                               // Determine distance for positioning command (relative)
                               IF (#configuration.jog.mode = #JOG_MODE_NEW_INCREMENT) // In this mode a new increment is always set
                                 OR ((#configuration.jog.mode = #JOG_MODE_CONTINUE_INCREMENT) AND (#statResetIncJog = TRUE))
                               THEN
                                 #statResetIncJog := FALSE;
                                 // New increment
                                 #statIncJogStartPosition := "LAxisCtrl_UnpubAxisPosition"(#statAxis); // Targetposition for increment
                                 #statIncrement := ABS(#configuration.jog.increment); // absolute Distance for increment
                                 IF (#statBasicCommand.%X2 = TRUE) THEN
                                   // JogForward selected
                                   #statPosition := ABS(#configuration.jog.increment);
                                   #statIncrement := #statPosition;
                                   #statIncJogDirectionOld := #FORWARD_DIR;
                                 ELSIF (#statBasicCommand.%X3 = TRUE) THEN
                                   // JogBackward selected
                                   #statPosition := - ABS(#configuration.jog.increment);
                                   #statIncrement := #statPosition;
                                   #statIncJogDirectionOld := #BACKWARD_DIR;
                                 ELSE
                                   // Normal not possible to reach ELSE-branch
                                   #statIncJogDirectionOld := 0;
                                 END_IF;
                               ELSE
                                 // Check for modulo axis
                                 IF ("LAxisCtrl_UnpubAxisModuloEnabled"(#statAxis) = FALSE) THEN
                                   // No Modulo enabled
                                   // Continue increment
                                   #statPosition := (#statIncJogStartPosition + #statIncrement) - "LAxisCtrl_UnpubAxisPosition"(#statAxis);
                                   // Distance   :=            setpoint                         - actualvalue
                                 ELSE
                                   // Modulo enabled
                                   #statPosition := #statIncJogDistance;
                                 END_IF;
                               END_IF;
                               #statIncJogSubState := #INC_JOG_START;

                               // Store Dynamics
                               #statBasicVelocity := ABS(#configuration.jog.velocity);
                               #statBasicAcceleration := #configuration.jog.acceleration;
                               #statBasicDeceleration := #configuration.jog.deceleration;
                               #statBasicJerk := #configuration.jog.jerk;
                             ELSE
                               // Errorhandling - Invalid direction (forward and backward selected)
                               #statStatus := #ERR_INVALID_JOG_DIR;
                               #statStatusText := STRING#'ERR_INVALID_JOG_DIR';
                               #statErrorAutoCleared := TRUE;
                               #statDiagnostics.subfunctionStatus := #statSubfunctionStatus := 0;
                               #statDiagnostics.basicMotionState := #statBasicMotionState;
                               // Set next state
                               #statFBState := #AXIS_STOP_ON_ERROR_SELECTION;
                               #statBasicMotionState := #NO_SELECTION;
                               #statExeOfBasicMotion := #CMD_ERROR;
                               #statIncJogSubState := #INC_JOG_IDLE;
                             END_IF;

                           ELSIF ((#statBasicCommand.%X2 = FALSE) AND (#statBasicCommand.%X3 = FALSE)) // No jog input selected --> Stop moving
                             AND (#statIncJogSubState <> #INC_JOG_STOP)
                           THEN
                             // Reset HALT command
                             #instHalt(Axis := #statAxis,
                                       Execute := FALSE);
                             #statIncJogSubState := #INC_JOG_STOP;
                             #statIncJogDistance := "LAxisCtrl_UnpubAxisPositioningDistance"(#statAxis);

                           ELSIF (#statBasicCommand.%X2 = TRUE) AND (#statBasicCommand.%X3 = TRUE) // jogForward and jogBackward selected - Error
                           THEN
                             // Reset HALT command
                             #instHalt(Axis := #statAxis,
                                       Execute := FALSE);
                             #statIncJogSubState := #INC_JOG_STOP;
                             // Errorhandling
                             #statStatus := #ERR_INVALID_JOG_DIR;
                             #statStatusText := STRING#'ERR_INVALID_JOG_DIR';
                             #statErrorAutoCleared := TRUE;
                             #statDiagnostics.subfunctionStatus := #statSubfunctionStatus := 0;
                             // Set next state
                             #statExeOfBasicMotion := #CMD_ERROR;
                             #statBasicMotionState := #NO_SELECTION;
                             #statFBState := #AXIS_STOP_ON_ERROR_SELECTION;
                           ELSE
                             ; // Command running
                           END_IF;

                           // Select motion
                           CASE #statIncJogSubState OF
                             #INC_JOG_IDLE:
                               ; // Do nothing - Error occurred (jogforward and jogbackward are set in firstCycle of operation)

                             #INC_JOG_START: // Run jog operation --> Motion stops automatically if increment complete
                               #instMoveRelative(Axis := #statAxis,
                                                 Execute := TRUE,
                                                 Distance := #statPosition,
                                                 Velocity := #statBasicVelocity,
                                                 Acceleration := #statBasicAcceleration,
                                                 Deceleration := #statBasicDeceleration,
                                                 Jerk := #statBasicJerk);

                               // Evaluate MC_Command
                               IF (#instMoveRelative.Done = TRUE) THEN
                                 // Increment completed
                                 #statResetIncJog := TRUE;
                                 // Set next state
                                 #statExeOfBasicMotion := #CMD_DONE;
                                 #statIncJogSubState := #INC_JOG_IDLE;

                               ELSIF (#instMoveRelative.Error = TRUE) THEN
                                 #statResetIncJog := TRUE;
                                 // Errorhandling
                                 #statStatus := #ERR_MC_MOVERELATIVE;
                                 #statStatusText := STRING#'ERR_MC_MOVERELATIVE';
                                 #statErrorAutoCleared := TRUE;
                                 #statDiagnostics.subfunctionStatus := #statSubfunctionStatus := #instMoveRelative.ErrorID;
                                 // Set next state
                                 #statFBState := #AXIS_STOP_ON_ERROR_SELECTION;
                                 #statBasicMotionState := #NO_SELECTION;
                                 #statExeOfBasicMotion := #CMD_ERROR;
                                 #statIncJogSubState := #INC_JOG_IDLE;

                               ELSIF (#instMoveRelative.CommandAborted = TRUE) THEN
                                 #statResetIncJog := TRUE;
                                 #statExeOfBasicMotion := #CMD_ABORTED;
                                 #statIncJogSubState := #INC_JOG_IDLE;
                               ELSE
                                 ; // Wait for next state
                               END_IF;

                             #INC_JOG_STOP: // Executed if inputs are reset --> Stop jog operation OR if jogForward and jogBackward are set --> Error and stop axis
                               #instHalt(Axis := #statAxis,
                                         Execute := TRUE,
                                         Deceleration := #statBasicDeceleration,
                                         AbortAcceleration := FALSE,
                                         Jerk := #statBasicJerk);

                               // Evaluate MC_Command
                               IF (#instHalt.Done = TRUE) THEN
                                 // Set next state
                                 #statExeOfBasicMotion := #CMD_END_PROCESS;
                                 #statIncJogSubState := #INC_JOG_IDLE;

                               ELSIF (#instHalt.Error = TRUE) THEN
                                 #statResetIncJog := TRUE;
                                 // Errorhandling
                                 #statStatus := #ERR_MC_HALT;
                                 #statStatusText := STRING#'ERR_MC_HALT';
                                 #statErrorAutoCleared := TRUE;
                                 #statDiagnostics.subfunctionStatus := #statSubfunctionStatus := #instHalt.ErrorID;
                                 // Set next state
                                 #statFBState := #AXIS_STOP_ON_ERROR_SELECTION;
                                 #statBasicMotionState := #NO_SELECTION;
                                 #statExeOfBasicMotion := #CMD_ERROR;
                                 #statIncJogSubState := #INC_JOG_IDLE;

                               ELSIF (#instHalt.CommandAborted = TRUE) THEN
                                 #statResetIncJog := TRUE;
                                 // Set next state
                                 #statIncJogSubState := #INC_JOG_IDLE;
                                 #statExeOfBasicMotion := #CMD_ABORTED;
                               ELSE
                                 ; // Wait for stopping axis
                               END_IF;
                             ELSE
                               // Errorhandling
                               #statStatus := #ERR_UNDEFINED_INCREMENTAL_JOG_SUBSTATE;
                               #statStatusText := STRING#'ERR_UNDEFINED_INCREMENTAL_JOG_SUBSTATE';
                               #statErrorUserCleared := TRUE;
                               #statDiagnostics.subfunctionStatus := #statSubfunctionStatus := 0;
                               // Set errorstate
                               #statFBState := #FB_ERROR;
                           END_CASE;

                         #CMD_DONE,
                         #CMD_ABORTED,
                         #CMD_ERROR,
                         #CMD_END_PROCESS:
                           // Return to NO_SELECTION if command finished
                           IF (#statBasicCommand.%X2 = FALSE) AND (#statBasicCommand.%X3 = FALSE)
                           THEN
                             // jogForward and jogbackward inputs are reset
                             #statExeOfBasicMotion := #CMD_BUSY;
                             #statBasicMotionState := #NO_SELECTION;
                           ELSE
                             ; // Wait for falling edge at inputs for jog
                           END_IF;
                         ELSE
                           // Errorhandling
                           #statStatus := #ERR_UNDEFINED_INCREMENTAL_JOG_STATE;
                           #statStatusText := STRING#'ERR_UNDEFINED_INCREMENTAL_JOG_STATE';
                           #statErrorUserCleared := TRUE;
                           #statDiagnostics.subfunctionStatus := #statSubfunctionStatus := 0;
                           #statDiagnostics.basicMotionState := #statBasicMotionState;
                           // Set errorstate
                           #statFBState := #FB_ERROR;
                       END_CASE;
                     END_REGION
                   ELSE
                     // Errorhandling - Invalid jog state
                     #statStatus := #ERR_INVALID_JOG_MODE;
                     #statStatusText := STRING#'#ERR_INVALID_JOG_MODE';
                     #statErrorAutoCleared := TRUE;
                     #statDiagnostics.subfunctionStatus := #statSubfunctionStatus := 0;
                     // Set next state
                     #statFBState := #AXIS_STOP_ON_ERROR_SELECTION;
                     #statBasicMotionState := #NO_SELECTION;
                 END_CASE;
               END_REGION

             #MOVE_VELOCITY_SELECTED:
               // Additional features (applicative): Change setpoint on the fly (Velocity) 
               REGION MOVEVELOCITY_SELECTED
                 // Firstcycle of command
                 IF (#statFirstCycleBasicMotion = TRUE) THEN
                   // Reset MC_MOVEVELOCITY command
                   #instMoveVelocity(Axis := #statAxis,
                                     Execute := FALSE);

                   #statVelocityChangeOnTheFly := #configuration.moveVelocity.velocityChangeOnTheFly;
                   #statBasicVelocity := #configuration.moveVelocity.velocity;                     // Store the last adjusted velocity value
                   #statBasicAcceleration := #configuration.moveVelocity.acceleration;             // Store the last adjusted acceleration value
                   #statBasicDeceleration := #configuration.moveVelocity.deceleration;             // Store the last adjusted deceleration value
                   #statBasicJerk := #configuration.moveVelocity.jerk;                             // Store the last adjusted jerk value 
                   #statDirection := #configuration.moveVelocity.direction;                        // Store the last adjusted axis direction 
                   #statPositionControlled := #configuration.moveVelocity.positionControlled;      // Store the last adjusted motion mode

                 ELSIF (#statVelocityChangeOnTheFly = TRUE) AND (#configuration.moveVelocity.velocity <> #statBasicVelocity) // Velocity changed
                   AND (#instMoveVelocity.CommandAborted = FALSE)
                 THEN
                   // Reset MC_MOVEVELOCITY command
                   #instMoveVelocity(Axis := #statAxis,
                                     Execute := FALSE);
                   #statBasicVelocity := #configuration.moveVelocity.velocity;                     // Store the last adjusted velocity value

                   // V1.0.5 Copy also dynamics
                   #statBasicAcceleration := #configuration.moveVelocity.acceleration;             // Store the last adjusted acceleration value
                   #statBasicDeceleration := #configuration.moveVelocity.deceleration;             // Store the last adjusted deceleration value
                   #statBasicJerk := #configuration.moveVelocity.jerk;                             // Store the last adjusted jerk value 
                   #statDirection := #configuration.moveVelocity.direction;                        // Store the last adjusted axis direction 
                   #statPositionControlled := #configuration.moveVelocity.positionControlled;      // Store the last adjusted motion mode
                 END_IF;

                 // Call MC_Command
                 #instMoveVelocity(Axis := #statAxis,
                                   Execute := #statBasicCommand.%X4 OR #statFirstCycleBasicMotion, // Input: moveVelocity
                                   Velocity := #statBasicVelocity,
                                   Acceleration := #statBasicAcceleration,
                                   Deceleration := #statBasicDeceleration,
                                   Jerk := #statBasicJerk,
                                   Direction := #statDirection,
                                   PositionControlled := #statPositionControlled,
                                   Current := FALSE);

                 // Evaluate MC_Command
                 IF (#instMoveVelocity.Busy = FALSE) AND
                   (#instMoveVelocity.Error = FALSE) AND
                   (#instMoveVelocity.CommandAborted = FALSE) AND
                   (#instMoveVelocity.InVelocity = FALSE)
                 THEN
                   // Return to NO_SELECTION if command finished
                   #statBasicMotionState := #NO_SELECTION;

                 ELSIF (#instMoveVelocity.Error = TRUE)
                 THEN
                   // Errorhandling
                   #statStatus := #ERR_MC_MOVEVELOCITY;
                   #statStatusText := STRING#'ERR_MC_MOVEVELOCITY';
                   #statErrorAutoCleared := TRUE;
                   #statDiagnostics.subfunctionStatus := #statSubfunctionStatus := #instMoveVelocity.ErrorID;
                   #statVelocityChangeOnTheFly := FALSE;
                   // Set next state
                   #statFBState := #AXIS_STOP_ON_ERROR_SELECTION;
                   #statBasicMotionState := #NO_SELECTION;
                 ELSE
                   ; // Command selected
                 END_IF;

                 // Write MC_Command outputs to internal variable
                 #statExeOfBasicMotion := 16#0;
                 #statExeOfBasicMotion.%X0 := #instMoveVelocity.Busy;
                 #statExeOfBasicMotion.%X2 := #instMoveVelocity.CommandAborted;
                 #statExeOfBasicMotion.%X3 := #instMoveVelocity.Error;
                 #statExeOfBasicMotion.%X4 := #instMoveVelocity.InVelocity;
               END_REGION

             #POS_RELATIVE_SELECTED:
               // Additional features (applicative): Specified direction
               REGION POS_RELATIVE_SELECTED
                 // Firstcycle of command
                 IF (#statFirstCycleBasicMotion = TRUE) THEN
                   // Configurate the direction of rotation
                   IF ((#configuration.posRelative.direction = 0) AND (#configuration.posRelative.distance >= 0.0)) // Sign of distance is evaluated
                     OR (#configuration.posRelative.direction = #FORWARD_DIR) // Forward direction
                   THEN
                     #statPosition := ABS(#configuration.posRelative.distance);
                     // Reset MC_MOVERELATIVE command
                     #instMoveRelative(Axis := #statAxis,
                                       Execute := FALSE);
                     #statApplicativeBasicMotionError := FALSE;

                   ELSIF ((#configuration.posRelative.direction = 0) AND (#configuration.posRelative.distance < 0.0)) // Sign of distance is evaluated
                     OR (#configuration.posRelative.direction = #BACKWARD_DIR) // Backward direction
                   THEN
                     #statPosition := - ABS(IN := #configuration.posRelative.distance);
                     // Reset MC_MOVERELATIVE command
                     #instMoveRelative(Axis := #statAxis,
                                       Execute := FALSE);
                     #statApplicativeBasicMotionError := FALSE;
                   ELSE
                     // Errorhandling - Invalid direction
                     #statStatus := #ERR_INVALID_POS_RELATIVE_DIR;
                     #statStatusText := STRING#'ERR_INVALID_POS_RELATIVE_DIR';
                     #statErrorAutoCleared := TRUE;
                     #statDiagnostics.subfunctionStatus := #statSubfunctionStatus := 0;
                     #statApplicativeBasicMotionError := TRUE;
                     // Set next state
                     #statFBState := #AXIS_STOP_ON_ERROR_SELECTION;
                     #statBasicMotionState := #NO_SELECTION;
                   END_IF;
                 END_IF;

                 IF (#statApplicativeBasicMotionError = FALSE) THEN
                   // Call MC_Command
                   #instMoveRelative(Axis := #statAxis,
                                     Execute := #statBasicCommand.%X5 OR #statFirstCycleBasicMotion, // Input: posRelative
                                     Distance := #statPosition,
                                     Velocity := #configuration.posRelative.velocity,
                                     Acceleration := #configuration.posRelative.acceleration,
                                     Deceleration := #configuration.posRelative.deceleration,
                                     Jerk := #configuration.posRelative.jerk);

                   // Evaluate MC_Command
                   IF (#instMoveRelative.Busy = FALSE) AND
                     (#instMoveRelative.Error = FALSE) AND
                     (#instMoveRelative.Done = FALSE) AND
                     (#instMoveRelative.CommandAborted = FALSE)
                   THEN
                     // Return to NO_SELECTION if command finished
                     #statBasicMotionState := #NO_SELECTION;

                   ELSIF (#instMoveRelative.Error = TRUE) THEN
                     // Errorhandling
                     #statStatus := #ERR_MC_MOVERELATIVE;
                     #statStatusText := STRING#'ERR_MC_MOVERELATIVE';
                     #statErrorAutoCleared := TRUE;
                     #statDiagnostics.subfunctionStatus := #statSubfunctionStatus := #instMoveRelative.ErrorID;
                     // Set next state
                     #statFBState := #AXIS_STOP_ON_ERROR_SELECTION;
                     #statBasicMotionState := #NO_SELECTION;
                   ELSE
                     ; // Command selected
                   END_IF;

                   // Write MC_Command outputs to internal variable
                   #statExeOfBasicMotion := 16#0;
                   #statExeOfBasicMotion.%X0 := #instMoveRelative.Busy;
                   #statExeOfBasicMotion.%X1 := #instMoveRelative.Done;
                   #statExeOfBasicMotion.%X2 := #instMoveRelative.CommandAborted;
                   #statExeOfBasicMotion.%X3 := #instMoveRelative.Error;
                 ELSE
                   ; // Direction not valid
                 END_IF;
               END_REGION

             #POS_ABSOLUTE_SELECTED:
               // Additional features (applicative): Change setpoint on the fly (Velocity and Position)
               REGION POS_ABSOLUTE_SELECTED
                 // Firstcycle of command
                 IF (#statFirstCycleBasicMotion = TRUE) THEN
                   // Reset MC_MOVEABSOLUTE command
                   #instMoveAbsolute(Axis := #statAxis,
                                     Execute := FALSE);
                   #statPosition := #configuration.posAbsolute.position;
                   #statBasicVelocity := #configuration.posAbsolute.velocity;         // Store the last adjusted velocity value
                   #statBasicAcceleration := #configuration.posAbsolute.acceleration; // Store the last adjusted accerlation value
                   #statBasicDeceleration := #configuration.posAbsolute.deceleration; // Store the last adjusted deceleration value
                   #statBasicJerk := #configuration.posAbsolute.jerk;                 // Store the last adjusted jerk value
                   #statDirection := #configuration.posAbsolute.direction;

                   #statVelocityChangeOnTheFly := #configuration.posAbsolute.velocityChangeOnTheFly;
                   #statPositionChangeOnTheFly := #configuration.posAbsolute.positionChangeOnTheFly;

                 ELSIF (((#statVelocityChangeOnTheFly = TRUE) AND (#configuration.posAbsolute.velocity <> #statBasicVelocity))
                   OR ((#statPositionChangeOnTheFly = TRUE) AND (#configuration.posAbsolute.position <> #statPosition)))
                   AND (#instMoveAbsolute.CommandAborted = FALSE)
                 THEN
                   #instMoveAbsolute(Axis := #statAxis,
                                     Execute := FALSE);

                   IF (#statVelocityChangeOnTheFly = TRUE) THEN // Apply the new velocity value
                     #statBasicVelocity := #configuration.posAbsolute.velocity;

                     // V1.0.5 Copy also dynamics
                     #statBasicAcceleration := #configuration.posAbsolute.acceleration;             // Store the last adjusted acceleration value
                     #statBasicDeceleration := #configuration.posAbsolute.deceleration;             // Store the last adjusted deceleration value
                     #statBasicJerk := #configuration.posAbsolute.jerk;                             // Store the last adjusted jerk value 
                     #statDirection := #configuration.posAbsolute.direction;                        // Store the last adjusted axis direction 
                   END_IF;

                   IF (#statPositionChangeOnTheFly = TRUE) THEN // Apply the new position value
                     #statPosition := #configuration.posAbsolute.position;

                     // V1.0.5 Copy also dynamics
                     #statBasicVelocity := #configuration.posAbsolute.velocity;
                     #statBasicAcceleration := #configuration.posAbsolute.acceleration;             // Store the last adjusted acceleration value
                     #statBasicDeceleration := #configuration.posAbsolute.deceleration;             // Store the last adjusted deceleration value
                     #statBasicJerk := #configuration.posAbsolute.jerk;                             // Store the last adjusted jerk value 
                     #statDirection := #configuration.posAbsolute.direction;                        // Store the last adjusted axis direction 
                   END_IF;

                   // Reset MC_MOVEABSOLUTE command
                   #instMoveAbsolute(Axis := #statAxis,
                                     Execute := FALSE);
                 END_IF;

                 #instMoveAbsolute(Axis := #statAxis,
                                   Execute := #statBasicCommand.%X6 OR #statFirstCycleBasicMotion, // Input: posAbsolute
                                   Position := #statPosition,
                                   Velocity := #statBasicVelocity,
                                   Acceleration := #statBasicAcceleration,
                                   Deceleration := #statBasicDeceleration,
                                   Jerk := #statBasicJerk,
                                   Direction := #statDirection);

                 // Evaluate MC_Command
                 IF (#instMoveAbsolute.Busy = FALSE) AND
                   (#instMoveAbsolute.Error = FALSE) AND
                   (#instMoveAbsolute.Done = FALSE) AND
                   (#instMoveAbsolute.CommandAborted = FALSE)
                 THEN
                   // Return to NO_SELECTION if command finished
                   #statBasicMotionState := #NO_SELECTION;

                 ELSIF (#instMoveAbsolute.Error = TRUE) THEN
                   // Errorhandling
                   #statStatus := #ERR_MC_MOVEABSOLUTE;
                   #statStatusText := STRING#'ERR_MC_MOVEABSOLUTE';
                   #statErrorAutoCleared := TRUE;
                   #statDiagnostics.subfunctionStatus := #statSubfunctionStatus := #instMoveAbsolute.ErrorID;
                   #statVelocityChangeOnTheFly := FALSE;
                   #statPositionChangeOnTheFly := FALSE;
                   // Set next state
                   #statFBState := #AXIS_STOP_ON_ERROR_SELECTION;
                   #statBasicMotionState := #NO_SELECTION;
                 ELSE
                   ; // Command selected
                 END_IF;

                 // Write MC_Command outputs to internal variable
                 #statExeOfBasicMotion := 16#0;
                 #statExeOfBasicMotion.%X0 := #instMoveAbsolute.Busy;
                 #statExeOfBasicMotion.%X1 := #instMoveAbsolute.Done;
                 #statExeOfBasicMotion.%X2 := #instMoveAbsolute.CommandAborted;
                 #statExeOfBasicMotion.%X3 := #instMoveAbsolute.Error;
               END_REGION

             #ACTIVE_HOMING_SELECTED:
               // Additional feature (applicative): homing on fixed stop
               REGION ACTIVE_HOMING_SELECTED
                 // Firstcycle of command
                 IF (#statFirstCycleBasicMotion = TRUE) THEN
                   #statActiveHomingState := #configuration.homing.extendedMode;
                   #statExeOfBasicMotion := #CMD_BUSY;
                   #statPassiveHomingState := #NO_HOMING_ACTIVE;
                 END_IF;
                 // Selection of extended homing mode  
                 CASE #statActiveHomingState OF
                   #STANDARD_HOMING:
                     // No additional features
                     REGION STANDARD_HOMING
                       // Firstcycle of command
                       IF (#statFirstCycleBasicMotion = TRUE) THEN
                         // Reset MC_HOME command
                         #instHome(Axis := #statAxis,
                                   Execute := FALSE);
                       END_IF;

                       // Call MC_Command
                       #instHome(Axis := #statAxis,
                                 Execute := #statBasicCommand.%X10 OR #statFirstCycleBasicMotion, // Input: homing
                                 Position := #configuration.homing.position,
                                 Mode := #configuration.homing.mode);

                       // Evaluate MC_Command
                       IF (#instHome.Busy = FALSE) AND
                         (#instHome.Done = FALSE) AND
                         (#instHome.CommandAborted = FALSE) AND
                         (#instHome.Error = FALSE)
                       THEN
                         // Return to NO_SELECTION if command finished
                         #statActiveHomingState := #STANDARD_HOMING;
                         #statBasicMotionState := #NO_SELECTION;

                       ELSIF (#instHome.Error = TRUE) THEN
                         // Errorhandling
                         #statStatus := #ERR_MC_HOME;
                         #statStatusText := STRING#'ERR_MC_HOME';
                         #statErrorAutoCleared := TRUE;
                         #statDiagnostics.subfunctionStatus := #statSubfunctionStatus := #instHome.ErrorID;
                         #statFBState := #AXIS_STOP_ON_ERROR_SELECTION;
                         #statBasicMotionState := #NO_SELECTION;
                       ELSE
                         ; // Command selected
                       END_IF;
                       #statExeOfBasicMotion := 16#0;
                       #statExeOfBasicMotion.%X0 := #instHome.Busy;
                       #statExeOfBasicMotion.%X1 := #instHome.Done;
                       #statExeOfBasicMotion.%X2 := #instHome.CommandAborted;
                       #statExeOfBasicMotion.%X3 := #instHome.Error;
                     END_REGION

                   #HOMING_ON_FIXED_STOP,
                   #HOMING_ON_FIXED_STOP_WITH_MOVING_OUT_OF_CLAMPING, // V1.0.5 New extended homing mode
                   #HOMING_ON_FIXED_STOP_WITH_MOVING_TO_TARGET_POSITION: // V1.2.0 new extended homing mode
                     // This case is additional feature (MC_MOVEVELOCITY and MC_HOME internal used)
                     REGION REFERENCE_TO_FIXED_STOP
                       CASE #statExeOfBasicMotion OF
                         #CMD_BUSY:
                           // Firstcycle of command
                           IF (#statFirstCycleBasicMotion = TRUE) THEN

                             // Read operative sensor
                             #tempIndex := UDINT_TO_INT("LAxisCtrl_UnpubAxisOperativeSensor"(axis := #statAxis));

                             IF (#tempIndex < 1) THEN
                               #tempIndex := 1;
                             END_IF;

                             IF ("LAxisCtrl_UnpubAxisHomingDirection"(axis := #statAxis, index := #tempIndex) = 0)
                             THEN
                               // Positive direction
                               #statDirection := #FORWARD_DIR;
                             ELSE
                               // Negative direction
                               #statDirection := #BACKWARD_DIR;
                             END_IF;

                             // Check if homing on fixed stop is allowed  
                             IF ("LAxisCtrl_UnpubAxisModuloEnabled"(#statAxis) = TRUE) THEN
                               // Modulo enabled - Errorhandling
                               #statStatus := #ERR_MODULO_NOT_ALLOWED;
                               #statStatusText := STRING#'ERR_MODULO_NOT_ALLOWED';
                               #statErrorAutoCleared := TRUE;
                               #statDiagnostics.subfunctionStatus := #statSubfunctionStatus := 0;
                               #statDiagnostics.basicMotionState := #statBasicMotionState;
                               // Set next state
                               #statFBState := #AXIS_STOP_ON_ERROR_SELECTION;
                               #statBasicMotionState := #NO_SELECTION;
                               #statActiveHomingState := #STANDARD_HOMING;
                               #statHomingSubState := #HOMING_IDLE;

                             ELSIF (#configuration.homing.extendedModeTorqueLimit = 0.0) // Torqueliming 0 in configuration 
                             THEN
                               // Errorhandling -  Torquevalue 0 configured
                               #statStatus := #ERR_INVALID_TORQUE_LIMIT;
                               #statStatusText := STRING#'ERR_INVALID_TORQUE_LIMIT';
                               #statErrorAutoCleared := TRUE;
                               #statDiagnostics.subfunctionStatus := #statSubfunctionStatus := 0;
                               #statDiagnostics.basicMotionState := #statBasicMotionState;
                               // Set next state
                               #statFBState := #AXIS_STOP_ON_ERROR_SELECTION;
                               #statBasicMotionState := #NO_SELECTION;
                               #statActiveHomingState := #STANDARD_HOMING;
                               #statHomingSubState := #HOMING_IDLE;

                             ELSIF ("LAxisCtrl_UnpubAxisReferencingVelocity"(#statAxis) = 0.0)
                             THEN
                               // Errorhandling -  Velocity 0 configured
                               #statStatus := #ERR_INVALID_VELOCITY;
                               #statStatusText := STRING#'ERR_INVALID_VELOCITY';
                               #statErrorAutoCleared := TRUE;
                               #statDiagnostics.subfunctionStatus := #statSubfunctionStatus := 0;
                               #statDiagnostics.basicMotionState := #statBasicMotionState;
                               // Set next state
                               #statFBState := #AXIS_STOP_ON_ERROR_SELECTION;
                               #statBasicMotionState := #NO_SELECTION;
                               #statActiveHomingState := #STANDARD_HOMING;
                               #statHomingSubState := #HOMING_IDLE;

                             ELSIF (#statActiveHomingState = #HOMING_ON_FIXED_STOP_WITH_MOVING_TO_TARGET_POSITION)
                               AND FALSE
                               OR (#configuration.homing.extendedModeTargetPosition > #configuration.homing.position) AND (#statDirection = #FORWARD_DIR)
                               OR (#configuration.homing.extendedModeTargetPosition < #configuration.homing.position) AND (#statDirection = #BACKWARD_DIR)
                             THEN
                               // Errorhandling -  Velocity 0 configured
                               #statStatus := #ERR_INVALID_TARGET_POSITION;
                               #statStatusText := STRING#'ERR_INVALID_TARGET_POSITION';
                               #statErrorAutoCleared := TRUE;
                               #statDiagnostics.subfunctionStatus := #statSubfunctionStatus := 0;
                               #statDiagnostics.basicMotionState := #statBasicMotionState;
                               // Set next state
                               #statFBState := #AXIS_STOP_ON_ERROR_SELECTION;
                               #statBasicMotionState := #NO_SELECTION;
                               #statActiveHomingState := #STANDARD_HOMING;
                               #statHomingSubState := #HOMING_IDLE;


                             ELSE
                               // Store dynamic values
                               #statHomingPosition := #configuration.homing.position;
                               #statBasicVelocity := "LAxisCtrl_UnpubAxisReferencingVelocity"(#statAxis);
                               #statBasicAcceleration := "LAxisCtrl_UnpubAxisDynamicDefaultAcc"(#statAxis);
                               #statBasicDeceleration := "LAxisCtrl_UnpubAxisDynamicDefaultDec"(#statAxis);
                               #statBasicJerk := "LAxisCtrl_UnpubAxisDynamicDefaultJerk"(#statAxis);
                               #statTorqueLimit := #configuration.homing.extendedModeTorqueLimit;

                               #statTorqueLimitingState := #FIXED_STOP_DETECTION_ACTIVE;
                               // Reset MC_Commands
                               #instHome(Axis := #statAxis,
                                         Execute := FALSE);
                               #instMoveVelocity(Axis := #statAxis,
                                                 Execute := FALSE);
                               #instMoveAbsolute(Axis := #statAxis,
                                                 Execute := FALSE);

                               // Determine the encoder type
                               IF ("LAxisCtrl_UnpubAxisSensorType"(axis := #statAxis, index := #tempIndex) = #INCREMENTAL_ENCODER) THEN
                                 #statHomingMode := #DIRECT_HOMING; // Direct homing (absolute)
                               ELSE
                                 #statHomingMode := #ABSOLUTE_ENCODER_ADJUSTMENT;
                               END_IF;
                               // Use always direct homing
                               //#statHomingMode := #DIRECT_HOMING; // Direct homing (absolute)
                               // Set next state
                               #statHomingSubState := #HOMING_FIXED_STOP_DETECTION;
                             END_IF;
                           END_IF;

                           // Call of subStateMachine
                           REPEAT
                             CASE #statHomingSubState OF
                               #HOMING_IDLE:
                                 #tempStateChangeActive := FALSE;
                                 // Do nothing, inserted no exectution of homing if error occurred in first cycle

                               #HOMING_FIXED_STOP_DETECTION:
                                 #tempStateChangeActive := FALSE;

                                 // Start axis to detect fixed stop
                                 #instMoveVelocity(Axis := #statAxis,
                                                   Execute := TRUE,
                                                   Velocity := #statBasicVelocity,
                                                   Acceleration := #statBasicAcceleration,
                                                   Deceleration := #statBasicDeceleration,
                                                   Jerk := #statBasicJerk,
                                                   PositionControlled := TRUE,
                                                   Direction := #statDirection);

                                 // Read Statusword
                                 #tempStatusWord := "LAxisCtrl_UnpubAxisStatusWord"(#statAxis);

                                 // Evaluate MC_Command
                                 IF (#tempStatusWord.%X30 = TRUE) THEN // inClamping = TRUE
                                   // Fixed stop detected --> start homing process
                                   #statHomingSubState := #HOMING_PROCESS;
                                   #tempStateChangeActive := TRUE;

                                 ELSIF (#instMoveVelocity.Error = TRUE) THEN
                                   // Errorhandling
                                   #statStatus := #ERR_MC_MOVEVELOCITY;
                                   #statStatusText := STRING#'ERR_MC_MOVEVELOCITY';
                                   #statErrorAutoCleared := TRUE;
                                   #statDiagnostics.subfunctionStatus := #statSubfunctionStatus := #instMoveVelocity.ErrorID;
                                   // Set next state
                                   #statFBState := #AXIS_STOP_ON_ERROR_SELECTION;
                                   #statBasicMotionState := #NO_SELECTION;
                                   #statActiveHomingState := #STANDARD_HOMING;
                                   #statExeOfBasicMotion := #CMD_ERROR;
                                   #statHomingSubState := #HOMING_IDLE;

                                 ELSIF (#instMoveVelocity.CommandAborted = TRUE) THEN
                                   // Set next state
                                   #statExeOfBasicMotion := #CMD_ABORTED;
                                   #statHomingSubState := #HOMING_IDLE;
                                 ELSE
                                   ;// Wait for detecting fixed stop
                                 END_IF;

                               #HOMING_PROCESS:
                                 #tempStateChangeActive := FALSE;
                                 // Execute MC_HOME
                                 #instHome(Axis := #statAxis,
                                           Execute := TRUE,
                                           Position := #statHomingPosition,
                                           Mode := #statHomingMode);

                                 // Evaluate MC_Command
                                 IF (#instHome.Done = TRUE) THEN
                                   // MC_HOME finished - Set next state
                                   #statHomingSubState := #HOMING_POSITION;
                                   #tempStateChangeActive := TRUE;

                                 ELSIF (#instHome.Error = TRUE) THEN
                                   // Errorhandling
                                   #statStatus := #ERR_MC_HOME;
                                   #statStatusText := STRING#'ERR_MC_HOME';
                                   #statErrorAutoCleared := TRUE;
                                   #statDiagnostics.subfunctionStatus := #statSubfunctionStatus := #instHome.ErrorID;
                                   // Set next state
                                   #statFBState := #AXIS_STOP_ON_ERROR_SELECTION;
                                   #statExeOfBasicMotion := #CMD_ERROR;
                                   #statHomingSubState := #HOMING_IDLE;

                                 ELSIF (#instHome.CommandAborted = TRUE) THEN
                                   // Set next state
                                   #statExeOfBasicMotion := #CMD_ABORTED;
                                   #statHomingSubState := #HOMING_IDLE;
                                 ELSE
                                   ;// Wait for finish homing process
                                 END_IF;

                               #HOMING_POSITION:
                                 #tempStateChangeActive := FALSE;
                                 CASE #statActiveHomingState OF
                                   #HOMING_ON_FIXED_STOP:
                                     // Execute moving to homeposition
                                     #instMoveAbsolute(Axis := #statAxis,
                                                       Execute := TRUE,
                                                       Position := #statHomingPosition,
                                                       Velocity := ABS(#statBasicVelocity),
                                                       Acceleration := #statBasicAcceleration,
                                                       Deceleration := #statBasicDeceleration,
                                                       Jerk := #statBasicJerk,
                                                       Direction := #SHORTEST_WAY_DIR);

                                     // Evaluate MC_Command
                                     IF (#instMoveAbsolute.Done = TRUE) THEN
                                       // Homeposition reached - Set next state
                                       #statExeOfBasicMotion := #CMD_DONE;
                                       #statHomingSubState := #HOMING_IDLE;

                                     ELSIF (#instMoveAbsolute.Error = TRUE) THEN
                                       // Errorhandling
                                       #statStatus := #ERR_MC_MOVEABSOLUTE;
                                       #statStatusText := STRING#'ERR_MC_MOVEABSOLUTE';
                                       #statErrorAutoCleared := TRUE;
                                       #statDiagnostics.subfunctionStatus := #statSubfunctionStatus := #instMoveAbsolute.ErrorID;
                                       // Set next state
                                       #statFBState := #AXIS_STOP_ON_ERROR_SELECTION;
                                       #statBasicMotionState := #CMD_BUSY;
                                       #statActiveHomingState := #STANDARD_HOMING;
                                       #statExeOfBasicMotion := #CMD_ERROR;
                                       #statHomingSubState := #HOMING_IDLE;

                                     ELSIF (#instMoveAbsolute.CommandAborted = TRUE) THEN
                                       // Set next state
                                       #statExeOfBasicMotion := #CMD_ABORTED;
                                       #statHomingSubState := #HOMING_IDLE;
                                     ELSE
                                       ; // Wait for reaching homeposition
                                     END_IF;

                                   #HOMING_ON_FIXED_STOP_WITH_MOVING_OUT_OF_CLAMPING: // V1.0.5 New extended homing mode
                                     // Execute moving to homeposition
                                     CASE #statDirection OF
                                       #FORWARD_DIR:
                                         #statHomingPosition -= (#DISTANCE_SCALING * "LAxisCtrl_UnpubAxisPositionTolerance"(#statAxis));

                                       #BACKWARD_DIR:
                                         #statHomingPosition += (#DISTANCE_SCALING * "LAxisCtrl_UnpubAxisPositionTolerance"(#statAxis));
                                     END_CASE;

                                     // Execute moving to homeposition
                                     #instMoveAbsolute(Axis := #statAxis,
                                                       Execute := TRUE,
                                                       Position := #statHomingPosition,
                                                       Velocity := ABS(#statBasicVelocity),
                                                       Acceleration := #statBasicAcceleration,
                                                       Deceleration := #statBasicDeceleration,
                                                       Jerk := #statBasicJerk,
                                                       Direction := #SHORTEST_WAY_DIR);

                                     // Evaluate MC_Command
                                     IF (#instMoveAbsolute.Done = TRUE) AND (#instTorqueLimiting.InClamping = FALSE)
                                     THEN
                                       // Homeposition reached - Set next state
                                       #statExeOfBasicMotion := #CMD_DONE;
                                       #statHomingSubState := #HOMING_IDLE;

                                     ELSIF (#instMoveAbsolute.Error = TRUE) THEN
                                       // Errorhandling
                                       #statStatus := #ERR_MC_MOVEABSOLUTE;
                                       #statStatusText := STRING#'ERR_MC_MOVEABSOLUTE';
                                       #statErrorAutoCleared := TRUE;
                                       #statDiagnostics.subfunctionStatus := #statSubfunctionStatus := #instMoveAbsolute.ErrorID;
                                       // Set next state
                                       #statFBState := #AXIS_STOP_ON_ERROR_SELECTION;
                                       #statBasicMotionState := #CMD_BUSY;
                                       #statActiveHomingState := #STANDARD_HOMING;
                                       #statExeOfBasicMotion := #CMD_ERROR;
                                       #statHomingSubState := #HOMING_IDLE;

                                     ELSIF (#instMoveAbsolute.CommandAborted = TRUE) THEN
                                       // Set next state
                                       #statExeOfBasicMotion := #CMD_ABORTED;
                                       #statHomingSubState := #HOMING_IDLE;

                                     ELSE
                                       ; // Wait for reaching homeposition
                                     END_IF;

                                   #HOMING_ON_FIXED_STOP_WITH_MOVING_TO_TARGET_POSITION: // V1.2.0 New extended homing mode
                                     // Execute moving to target position
                                     #instMoveAbsolute(Axis := #statAxis,
                                                       Execute := TRUE,
                                                       Position := #configuration.homing.extendedModeTargetPosition,
                                                       Velocity := ABS(#statBasicVelocity),
                                                       Acceleration := #statBasicAcceleration,
                                                       Deceleration := #statBasicDeceleration,
                                                       Jerk := #statBasicJerk);

                                     // Evaluate MC_Command
                                     IF (#instMoveAbsolute.Done = TRUE) AND (#instTorqueLimiting.InClamping = FALSE)
                                     THEN
                                       // Homeposition reached - Set next state
                                       #statExeOfBasicMotion := #CMD_DONE;
                                       #statHomingSubState := #HOMING_IDLE;

                                     ELSIF (#instMoveAbsolute.Error = TRUE) THEN
                                       // Errorhandling
                                       #statStatus := #ERR_MC_MOVEABSOLUTE;
                                       #statStatusText := STRING#'ERR_MC_MOVEABSOLUTE';
                                       #statErrorAutoCleared := TRUE;
                                       #statDiagnostics.subfunctionStatus := #statSubfunctionStatus := #instMoveAbsolute.ErrorID;
                                       // Set next state
                                       #statFBState := #AXIS_STOP_ON_ERROR_SELECTION;
                                       #statBasicMotionState := #CMD_BUSY;
                                       #statActiveHomingState := #STANDARD_HOMING;
                                       #statExeOfBasicMotion := #CMD_ERROR;
                                       #statHomingSubState := #HOMING_IDLE;

                                     ELSIF (#instMoveAbsolute.CommandAborted = TRUE) THEN
                                       // Set next state
                                       #statExeOfBasicMotion := #CMD_ABORTED;
                                       #statHomingSubState := #HOMING_IDLE;

                                     ELSE
                                       ; // Wait for reaching homeposition
                                     END_IF;
                                 END_CASE;
                               ELSE
                                 // Errorhandling 
                                 #statStatus := #ERR_UNDEFINED_EXTENDED_HOMING_SUBSTATE;
                                 #statStatusText := STRING#'ERR_UNDEFINED_EXTENDED_HOMING_SUBSTATE';
                                 #statErrorUserCleared := TRUE;
                                 #statDiagnostics.subfunctionStatus := #statSubfunctionStatus := 0;
                                 // Set errorstate
                                 #statFBState := #FB_ERROR;
                                 #tempStateChangeActive := FALSE;
                             END_CASE;

                           UNTIL (#tempStateChangeActive = FALSE) // Repeat execution if a state is changing
                           END_REPEAT;

                         #CMD_DONE,
                         #CMD_ABORTED,
                         #CMD_ERROR:
                           // Return to NO_SELECTION if command finished
                           IF (#statBasicCommand.%X10 = FALSE) // homing = FALSE
                           THEN
                             // Return to NO_HOMING_ACTIVE if command finished
                             #statBasicMotionState := #NO_SELECTION;
                             #statActiveHomingState := #STANDARD_HOMING;
                             #statExeOfBasicMotion := #CMD_BUSY;
                             #statHomingSubState := #HOMING_IDLE;
                           ELSE
                             ; // Wait for falling edge at homing command
                           END_IF;
                         ELSE
                           // Errorhandling
                           #statStatus := #ERR_UNDEFINED_EXTENDED_HOMING_STATE;
                           #statStatusText := STRING#'ERR_UNDEFINED_EXTENDED_HOMING_STATE';
                           #statErrorUserCleared := TRUE;
                           #statDiagnostics.subfunctionStatus := #statSubfunctionStatus := 0;
                           // Set errorstate
                           #statFBState := #FB_ERROR;
                       END_CASE;
                     END_REGION

                   ELSE
                     // Errorhandling
                     #statStatus := #ERR_INVALID_HOMING_EXTENDED_MODE;
                     #statStatusText := STRING#'ERR_INVALID_HOMING_EXTENDED_MODE';
                     #statErrorAutoCleared := TRUE;
                     #statDiagnostics.subfunctionStatus := #statSubfunctionStatus := 0;
                     // Set next state
                     #statFBState := #AXIS_STOP_ON_ERROR_SELECTION;
                     #statBasicMotionState := #NO_SELECTION;
                     #statActiveHomingState := #STANDARD_HOMING;
                     #statBasicMotionState := #NO_SELECTION;
                 END_CASE;
               END_REGION

             #GEAR_IN_RELATIVE_SELECTED:
               // Additional features (applicative): Change setpoint on the fly (gear ratio)
               REGION GEAR_IN_RELATIVE_SELECTED
                 // Firstcycle of command
                 IF (#statFirstCycleBasicMotion = TRUE) THEN
                   // Reset GEAR_IN command 
                   #instGearIn(Master := #master,
                               Slave := #statAxis,
                               Execute := FALSE);

                   #statRatioNumerator := #configuration.gearInRelative.ratioNumerator;
                   #statRatioDenominator := #configuration.gearInRelative.ratioDenominator;
                   #statBasicAcceleration := #configuration.gearInRelative.acceleration;
                   #statBasicDeceleration := #configuration.gearInRelative.deceleration;
                   #statBasicJerk := #configuration.gearInRelative.jerk;
                   #statRatioChangeOnTheFly := #configuration.gearInRelative.ratioChangeOnTheFly;

                 ELSIF ((#statRatioChangeOnTheFly = TRUE) // Flying change of ratio numerator
                   AND ((#configuration.gearInRelative.ratioNumerator <> #statRatioNumerator)
                   OR (#configuration.gearInRelative.ratioDenominator <> #statRatioDenominator)))
                   AND
                   (#instGearIn.CommandAborted = FALSE)
                 THEN
                   #instGearIn(Master := #master,
                               Slave := #statAxis,
                               Execute := FALSE);

                   #statRatioNumerator := #configuration.gearInRelative.ratioNumerator;   // Apply the new gear ratio numerator
                   #statRatioDenominator := #configuration.gearInRelative.ratioDenominator; // Apply the new gear ratio denominator

                   // V1.0.5 Copy also dynamics
                   #statBasicAcceleration := #configuration.gearInRelative.acceleration;
                   #statBasicDeceleration := #configuration.gearInRelative.deceleration;
                   #statBasicJerk := #configuration.gearInRelative.jerk;
                 END_IF;

                 // Call MC_Command
                 #instGearIn(Master := #master,
                             Slave := #statAxis,
                             Execute := #statBasicCommand.%X7 OR #statFirstCycleBasicMotion, // Input: gearInRelative
                             RatioNumerator := #statRatioNumerator,
                             RatioDenominator := #statRatioDenominator,
                             Acceleration := #statBasicAcceleration,
                             Deceleration := #statBasicDeceleration,
                             Jerk := #statBasicJerk);

                 // Evaluate MC_Command
                 IF (#instGearIn.Busy = FALSE) AND
                   (#instGearIn.Error = FALSE) AND
                   (#instGearIn.CommandAborted = FALSE) AND
                   (#instGearIn.InGear = FALSE)
                 THEN
                   // Return to NO_SELECTION if command finished
                   #statBasicMotionState := #NO_SELECTION;

                 ELSIF (#instGearIn.Error = TRUE) THEN
                   // Errorhandling
                   #statStatus := #ERR_MC_GEARIN;
                   #statStatusText := STRING#'ERR_MC_GEARIN';
                   #statErrorAutoCleared := TRUE;
                   #statDiagnostics.subfunctionStatus := #statSubfunctionStatus := #instGearIn.ErrorID;
                   #statRatioChangeOnTheFly := FALSE;
                   // Set next state
                   #statFBState := #AXIS_STOP_ON_ERROR_SELECTION;
                   #statBasicMotionState := #NO_SELECTION;
                 ELSE
                   ; // Command selected
                 END_IF;

                 // Write MC_Command outputs to internal variable
                 #statExeOfBasicMotion := 16#0;
                 #statExeOfBasicMotion.%X0 := #instGearIn.Busy;
                 #statExeOfBasicMotion.%X2 := #instGearIn.CommandAborted;
                 #statExeOfBasicMotion.%X3 := #instGearIn.Error;
                 //#statExeOfBasicMotion.%X6 := #tempStatusWord.%X21 AND NOT #instGearIn.InGear; // write Synchronizing only when bit of instance of MC_GearIn.InGear = FALSE
                 #statExeOfBasicMotion.%X7 := #instGearIn.InGear;
               END_REGION

             #GEAR_IN_ABSOLUTE_SELECTED:
               // Additional features (applicative): Change setpoint on the fly (gear ratio)
               REGION GEAR_IN_SELECTED
                 // Firstcycle of command
                 IF (#statFirstCycleBasicMotion = TRUE) THEN
                   // Reset GEAR_IN_POS command 
                   #instGearInPos(Master := #master,
                                  Slave := #statAxis,
                                  Execute := FALSE);

                   #statRatioNumerator := #configuration.gearInAbsolute.ratioNumerator;
                   #statRatioDenominator := #configuration.gearInAbsolute.ratioDenominator;
                   #statMasterSyncPosition := #configuration.gearInAbsolute.masterSyncPosition;
                   #statSlaveSyncPosition := #configuration.gearInAbsolute.slaveSyncPosition;
                   #statBasicSyncProfileReference := #configuration.gearInAbsolute.syncProfileReference;
                   #statBasicMasterStartDistance := #configuration.gearInAbsolute.masterStartDistance;
                   #statBasicVelocity := #configuration.gearInAbsolute.velocity;
                   #statBasicAcceleration := #configuration.gearInAbsolute.acceleration;
                   #statBasicDeceleration := #configuration.gearInAbsolute.deceleration;
                   #statBasicJerk := #configuration.gearInAbsolute.jerk;
                   #statBasicSyncDirection := #configuration.gearInAbsolute.syncDirection;
                   #statRatioChangeOnTheFly := #configuration.gearInAbsolute.ratioChangeOnTheFly;

                 ELSIF (((#statRatioChangeOnTheFly = TRUE) AND (#configuration.gearInAbsolute.ratioNumerator <> #statRatioNumerator))
                   OR ((#statRatioChangeOnTheFly = TRUE) AND (#configuration.gearInAbsolute.ratioDenominator <> #statRatioDenominator)))
                   AND
                   (#instGearInPos.CommandAborted = FALSE)
                 THEN
                   #instGearInPos(Master := #master,
                                  Slave := #statAxis,
                                  Execute := FALSE);

                   #statRatioNumerator := #configuration.gearInAbsolute.ratioNumerator;   // Apply the new gear ratio numerator
                   #statRatioDenominator := #configuration.gearInAbsolute.ratioDenominator; // Apply the new gear ratio denominator

                   // V1.0.5 Copy also dynamics
                   #statMasterSyncPosition := #configuration.gearInAbsolute.masterSyncPosition;
                   #statSlaveSyncPosition := #configuration.gearInAbsolute.slaveSyncPosition;
                   #statBasicSyncProfileReference := #configuration.gearInAbsolute.syncProfileReference;
                   #statBasicMasterStartDistance := #configuration.gearInAbsolute.masterStartDistance;
                   #statBasicVelocity := #configuration.gearInAbsolute.velocity;
                   #statBasicAcceleration := #configuration.gearInAbsolute.acceleration;
                   #statBasicDeceleration := #configuration.gearInAbsolute.deceleration;
                   #statBasicJerk := #configuration.gearInAbsolute.jerk;
                   #statBasicSyncDirection := #configuration.gearInAbsolute.syncDirection;
                 END_IF;

                 // Call MC_Command
                 #instGearInPos(Master := #master,
                                Slave := #statAxis,
                                Execute := #statBasicCommand.%X8 OR #statFirstCycleBasicMotion, // Input: gearInAbsolute
                                RatioNumerator := #statRatioNumerator,
                                RatioDenominator := #statRatioDenominator,
                                MasterSyncPosition := #statMasterSyncPosition,
                                SlaveSyncPosition := #statSlaveSyncPosition,
                                SyncProfileReference := #statBasicSyncProfileReference,
                                MasterStartDistance := #statBasicMasterStartDistance,
                                Velocity := #statBasicVelocity,
                                Acceleration := #statBasicAcceleration,
                                Deceleration := #statBasicDeceleration,
                                Jerk := #statBasicJerk,
                                SyncDirection := #statBasicSyncDirection);

                 // Evaluate MC_Command
                 IF (#instGearInPos.Busy = FALSE) AND
                   (#instGearInPos.Error = FALSE) AND
                   (#instGearInPos.CommandAborted = FALSE) AND
                   (#instGearInPos.StartSync = FALSE) AND
                   (#instGearInPos.InSync = FALSE)
                 THEN
                   // Return to NO_SELECTION if command finished
                   #statBasicMotionState := #NO_SELECTION;

                 ELSIF (#instGearInPos.Error = TRUE) THEN
                   // Errorhandling
                   #statStatus := #ERR_MC_GEARINPOS;
                   #statStatusText := STRING#'ERR_MC_GEARINPOS';
                   #statErrorAutoCleared := TRUE;
                   #statDiagnostics.subfunctionStatus := #statSubfunctionStatus := #instGearInPos.ErrorID;
                   #statRatioChangeOnTheFly := FALSE;
                   // Set next state
                   #statFBState := #AXIS_STOP_ON_ERROR_SELECTION;
                   #statBasicMotionState := #NO_SELECTION;
                 ELSE
                   ; // Command selected
                 END_IF;

                 // Write MC_Command outputs to internal variable
                 #statExeOfBasicMotion := 16#0;
                 #statExeOfBasicMotion.%X0 := #instGearInPos.Busy;
                 #statExeOfBasicMotion.%X2 := #instGearInPos.CommandAborted;
                 #statExeOfBasicMotion.%X3 := #instGearInPos.Error;
                 #statExeOfBasicMotion.%X6 := #instGearInPos.StartSync;
                 #statExeOfBasicMotion.%X7 := #instGearInPos.InSync;
               END_REGION

             #CAM_IN_SELECTED:
               REGION CAM_IN_SELECTED
                 // Firstcycle of command
                 IF (#statFirstCycleBasicMotion = TRUE) THEN
                   #statCam := #cam;
                   // Reset CAM_IN command 
                   #instCamIn(Master := #master,
                              Slave := #statAxis,
                              Cam := #statCam,
                              Execute := FALSE);

                   #statApplicationMode := #configuration.camIn.applicationMode;
                 END_IF;

                 // Call MC_Command
                 #instCamIn(Master := #master,
                            Slave := #statAxis,
                            Cam := #statCam,
                            Execute := #statBasicCommand.%X9 OR #statFirstCycleBasicMotion, // Input: camIn
                            MasterOffset := #configuration.camIn.masterOffset,
                            SlaveOffset := #configuration.camIn.slaveOffset,
                            MasterScaling := #configuration.camIn.masterScaling,
                            SlaveScaling := #configuration.camIn.slaveScaling,
                            MasterSyncPosition := #configuration.camIn.masterSyncPosition,
                            SyncProfileReference := #configuration.camIn.syncProfileReference,
                            MasterStartDistance := #configuration.camIn.masterStartDistance,
                            Velocity := #configuration.camIn.velocity,
                            Acceleration := #configuration.camIn.acceleration,
                            Deceleration := #configuration.camIn.deceleration,
                            Jerk := #configuration.camIn.jerk,
                            ApplicationMode := #configuration.camIn.applicationMode,
                            SyncDirection := #configuration.camIn.syncDirection);

                 // Evaluate MC_Command
                 IF ((#instCamIn.Busy = FALSE) AND
                   (#instCamIn.Error = FALSE) AND
                   (#instCamIn.CommandAborted = FALSE) AND
                   (#instCamIn.InSync = FALSE) AND
                   (#instCamIn.StartSync = FALSE) AND
                   (#statBasicCommand.%X9 = FALSE))
                   AND // V1.0.2 Wait for one cycle EndOfProfile (--> Done) before function is finished at applicationMode ONCE
                   ((#statApplicationMode <> #APPLICATION_MODE_ONCE) OR
                   ((#statApplicationMode = #APPLICATION_MODE_ONCE) AND (#instCamIn.EndOfProfile = FALSE)))
                 THEN
                   // Return to NO_SELECTION if command finished
                   #statBasicMotionState := #NO_SELECTION;

                 ELSIF (#instCamIn.Error = TRUE) THEN
                   // Errorhandling
                   #statStatus := #ERR_MC_CAMIN;
                   #statStatusText := STRING#'ERR_MC_CAMIN';
                   #statErrorAutoCleared := TRUE;
                   #statDiagnostics.subfunctionStatus := #statSubfunctionStatus := #instCamIn.ErrorID;
                   #statDiagnostics.basicMotionState := #statBasicMotionState;
                   #statFBState := #AXIS_STOP_ON_ERROR_SELECTION;
                   #statBasicMotionState := #NO_SELECTION;
                 ELSE
                   ; // Command selected
                 END_IF;

                 // Write MC_Command outputs to internal variable
                 #statExeOfBasicMotion := 16#0;
                 #statExeOfBasicMotion.%X0 := #instCamIn.Busy;
                 IF (#statApplicationMode = #APPLICATION_MODE_ONCE)
                 THEN
                   #statExeOfBasicMotion.%X1 := #instCamIn.EndOfProfile;
                 END_IF;
                 #statExeOfBasicMotion.%X2 := #instCamIn.CommandAborted;
                 #statExeOfBasicMotion.%X3 := #instCamIn.Error;
                 #statExeOfBasicMotion.%X6 := #instCamIn.StartSync;
                 #statExeOfBasicMotion.%X7 := #instCamIn.InSync;
                 #statExeOfBasicMotion.%X8 := #instCamIn.EndOfProfile;
               END_REGION

             #GEAR_OUT_CAM_OUT_SELECTED:
               REGION GEAR_AND_CAM_OUT_SELECTED
                 // Firstcycle of command
                 IF (#statFirstCycleBasicMotion = TRUE) THEN
                   #statApplicativeBasicMotionError := FALSE;
                   #statFirstCycleBasicMotion := FALSE;

                   // Reset CAM_OUT command 
                   #instCamOut(Slave := #statAxis,
                               Execute := FALSE,
                               SlavePosition := #configuration.gearOutCamOut.slavePosition,
                               SyncProfileReference := #configuration.gearOutCamOut.syncProfileReference,
                               MasterStopDistance := #configuration.gearOutCamOut.masterStopDistance,
                               Deceleration := #configuration.gearOutCamOut.deceleration,
                               Jerk := #configuration.gearOutCamOut.jerk,
                               SyncOutDirection := #configuration.gearOutCamOut.syncOutDirection);

                   // Reset GEAR_OUT command 
                   #instGearOut(Slave := #statAxis,
                                Execute := FALSE,
                                SlavePosition := #configuration.gearOutCamOut.slavePosition,
                                SyncProfileReference := #configuration.gearOutCamOut.syncProfileReference,
                                MasterStopDistance := #configuration.gearOutCamOut.masterStopDistance,
                                Deceleration := #configuration.gearOutCamOut.deceleration,
                                Jerk := #configuration.gearOutCamOut.jerk,
                                SyncOutDirection := #configuration.gearOutCamOut.syncOutDirection);

                   CASE #configuration.gearOutCamOut.gearOutCamOutMode OF
                     #SYNCOUT_MODE_AUTOMATIC,
                     #SYNCOUT_MODE_GEAROUT,
                     #SYNCOUT_MODE_CAMOUT:
                       // Get axis waiting function state V1.2.0
                       IF (#statTypeAxis = #SYNC_AXIS) THEN
                         IF (#statWaitingFunctionStateAbortAutomatic < 0) // < 0: Automatic abort of waiting sync commands disabled
                         THEN
                           // Read waiting function state of axis
                           #statWaitingFunctionState := "LAxisCtrl_UnpubWaitingFunctionStateSyncAxis"(#statAxis);
                         ELSE
                           // Waiting function state already read out
                           #statWaitingFunctionState := #statWaitingFunctionStateAbortAutomatic;
                         END_IF;
                         // Read function state of axis
                         #statFunctionState := "LAxisCtrl_UnpubFunctionStateSyncAxis"(#statAxis);
                       END_IF;

                       #statGearAndCamOutMode := #configuration.gearOutCamOut.gearOutCamOutMode;
                       #statSyncOutState := #SYNCOUT_STATE_CHECK_WAITING; // Set next state

                     ELSE
                       // Errorhandling - Invalid mode
                       #statStatus := #ERR_INVALID_GEAROUT_CAMOUT_MODE;
                       #statStatusText := STRING#'ERR_INVALID_GEAROUT_CAMOUT_MODE';
                       #statErrorAutoCleared := TRUE;
                       #statDiagnostics.subfunctionStatus := #statSubfunctionStatus := 0;
                       #statApplicativeBasicMotionError := TRUE;
                       // Set next state
                       #statFBState := #AXIS_STOP_ON_ERROR_SELECTION;
                       #statBasicMotionState := #NO_SELECTION;
                   END_CASE;
                 END_IF;

                 IF (#statApplicativeBasicMotionError = FALSE) THEN
                   CASE #statSyncOutState OF
                       // ===========================================================
                     #SYNCOUT_STATE_CHECK_WAITING:
                       REGION CHECK_WAITING_FUNCTION_STATE
                         CASE #statGearAndCamOutMode OF
                           #SYNCOUT_MODE_GEAROUT:
                             CASE #statWaitingFunctionStateAbortAutomatic OF
                               #WFS_FS_CAMIN:
                                 // Abort waiting camming in advance
                                 #instCamOut.SyncProfileReference := #CANCEL_ONLY_WAITING_GEARING_CAMMING;
                                 #statSyncOutState := #SYNCOUT_STATE_CAMOUT_WAITING_BUSY; // Set next state

                               #WFS_FS_GEARINPOS:
                                 CASE #configuration.gearOutCamOut.syncProfileReference OF
                                   #CANCEL_ONLY_WAITING_GEARING_CAMMING:
                                     // Only gearOut - Set next state
                                     #statSyncOutState := #SYNCOUT_STATE_CHECK_ACTIVE;
                                   ELSE
                                     CASE #statFunctionState OF
                                       #WFS_FS_GEARIN,
                                       #WFS_FS_GEARINPOS:
                                         // Active gearing function
                                         #statSyncOutState := #SYNCOUT_STATE_CHECK_ACTIVE; // Set next state
                                       ELSE
                                         // Abort waiting gearing in advance
                                         #instGearOut.SyncProfileReference := #CANCEL_ONLY_WAITING_GEARING_CAMMING;
                                         #statSyncOutState := #SYNCOUT_STATE_GEAROUT_WAITING_BUSY; // Set next state
                                     END_CASE;
                                 END_CASE;

                               ELSE
                                 // Only gearOut - Set next state
                                 #statSyncOutState := #SYNCOUT_STATE_CHECK_ACTIVE;
                             END_CASE;

                           #SYNCOUT_MODE_CAMOUT:
                             CASE #statWaitingFunctionStateAbortAutomatic OF
                               #WFS_FS_GEARINPOS: // Waiting
                                 // Abort waiting gearing in advance
                                 #instGearOut.SyncProfileReference := #CANCEL_ONLY_WAITING_GEARING_CAMMING;
                                 #statSyncOutState := #SYNCOUT_STATE_GEAROUT_WAITING_BUSY; // Set next state

                               #WFS_FS_CAMIN: // Waiting
                                 CASE #configuration.gearOutCamOut.syncProfileReference OF
                                   #CANCEL_ONLY_WAITING_GEARING_CAMMING:
                                     // Only gearOut - Set next state
                                     #statSyncOutState := #SYNCOUT_STATE_CHECK_ACTIVE;
                                   ELSE
                                     CASE #statFunctionState OF
                                       #WFS_FS_CAMIN: // Active
                                         #statSyncOutState := #SYNCOUT_STATE_CHECK_ACTIVE; // Set next state
                                       ELSE
                                         // Abort waiting gearing in advance
                                         #instGearOut.SyncProfileReference := #CANCEL_ONLY_WAITING_GEARING_CAMMING;
                                         #statSyncOutState := #SYNCOUT_STATE_CAMOUT_WAITING_BUSY; // Set next state
                                     END_CASE;
                                 END_CASE;
                               ELSE
                                 // Only camOut - Set next state
                                 #statSyncOutState := #SYNCOUT_STATE_CHECK_ACTIVE;
                             END_CASE;

                           #SYNCOUT_MODE_AUTOMATIC:
                             CASE #statWaitingFunctionState OF
                               #WFS_FS_GEARINPOS, // Waiting
                               #WFS_FS_GEAROUT: // Waiting
                                 CASE #statFunctionState OF
                                   #WFS_FS_GEARIN, // Active
                                   #WFS_FS_GEARINPOS: // Active
                                     ; // Gearing active - Waiting gearInPos will be aborted with MC_GEAROUT

                                   #WFS_FS_GEAROUT:
                                     IF (#statWaitingFunctionStateAbortAutomatic < 0) THEN
                                       ; // Automatic abort of waiting sync commands disabled
                                     ELSE
                                       // Automatic abort of waiting sync commands enabled - Separate call of MC_GearOut instruction is required
                                       #instGearOut.SyncProfileReference := #CANCEL_ONLY_WAITING_GEARING_CAMMING;
                                     END_IF;
                                   ELSE
                                     #instGearOut.SyncProfileReference := #CANCEL_ONLY_WAITING_GEARING_CAMMING;
                                 END_CASE;
                                 #statFunctionState := -1;// Function state has to be updated at next use
                                 #statSyncOutState := #SYNCOUT_STATE_GEAROUT_WAITING_BUSY; // Set next state

                               #WFS_FS_CAMIN,  // Waiting
                               #WFS_FS_CAMOUT:  // Waiting
                                 CASE #statFunctionState OF
                                   #WFS_FS_CAMIN: // Active
                                     ; // CamIn Active - Waiting CamIn will be aborted with MC_CAMOUT

                                   #WFS_FS_CAMOUT: // Active
                                     IF (#statWaitingFunctionStateAbortAutomatic < 0) THEN
                                       ; // Automatic abort of waiting sync commands disabled
                                     ELSE
                                       // Automatic abort of waiting sync commands enabled - Separate call of MC_CamOut instruction is required
                                       #instCamOut.SyncProfileReference := #CANCEL_ONLY_WAITING_GEARING_CAMMING;
                                     END_IF;
                                   ELSE
                                     #instCamOut.SyncProfileReference := #CANCEL_ONLY_WAITING_GEARING_CAMMING;
                                 END_CASE;
                                 #statFunctionState := -1;// Function state has to be updated at next use
                                 #statSyncOutState := #SYNCOUT_STATE_CAMOUT_WAITING_BUSY; // Set next state 

                               ELSE
                                 // No waiting synchronous operation
                                 #statSyncOutState := #SYNCOUT_STATE_CHECK_ACTIVE; // Set next state 
                             END_CASE;
                         END_CASE;
                         #tempStateChangeActive := TRUE;
                       END_REGION

                       // ===========================================================
                     #SYNCOUT_STATE_CHECK_ACTIVE:
                       REGION CHECK_ACTIVE_FUNCTION_STATE
                         #instGearOut.SyncProfileReference :=
                         #instCamOut.SyncProfileReference := #configuration.gearOutCamOut.syncProfileReference;

                         CASE #statGearAndCamOutMode OF
                           #SYNCOUT_MODE_GEAROUT:
                             #statSyncOutState := #SYNCOUT_STATE_GEAROUT_ACTIVE_BUSY; // Set next state

                           #SYNCOUT_MODE_CAMOUT:
                             #statSyncOutState := #SYNCOUT_STATE_CAMOUT_ACTIVE_BUSY; // Set next state

                           #SYNCOUT_MODE_AUTOMATIC:
                             CASE #configuration.gearOutCamOut.syncProfileReference OF
                               #CANCEL_ONLY_WAITING_GEARING_CAMMING:
                                 // No active synchronous operation
                                 #statSyncOutState := #SYNCOUT_STATE_DONE; // Set next state
                               ELSE
                                 // Update function state of axis
                                 IF (#statTypeAxis = #SYNC_AXIS) THEN
                                   IF (#statFunctionState < 0) THEN
                                     #statFunctionState := "LAxisCtrl_UnpubFunctionStateSyncAxis"(#statAxis);
                                   END_IF;
                                 END_IF;

                                 CASE #statFunctionState OF
                                   #WFS_FS_GEAROUT,   // Active - Leads to error of MC_Instruction
                                   #WFS_FS_GEARIN,    // Active
                                   #WFS_FS_GEARINPOS: // Active
                                     // Active gearing function
                                     #statSyncOutState := #SYNCOUT_STATE_GEAROUT_ACTIVE_BUSY; // Set next state

                                   #WFS_FS_CAMOUT, // Active - Leads to error of MC_Instruction
                                   #WFS_FS_CAMIN:  // Active
                                     // Active camming function
                                     #statSyncOutState := #SYNCOUT_STATE_CAMOUT_ACTIVE_BUSY; // Set next state

                                   ELSE
                                     // No active synchronous operation
                                     #statSyncOutState := #SYNCOUT_STATE_DONE; // Set next state
                                 END_CASE;
                             END_CASE;

                         END_CASE;
                         #tempStateChangeActive := TRUE;
                       END_REGION

                       // ===========================================================
                     #SYNCOUT_STATE_GEAROUT_WAITING_BUSY,
                     #SYNCOUT_STATE_GEAROUT_ACTIVE_BUSY:
                       REGION GEAROUT_BUSY
                         // Call MC_Instruction
                         #instGearOut(Slave := #statAxis,
                                      Execute := TRUE);

                         IF #instGearOut.Done THEN
                           CASE #statSyncOutState OF
                             #SYNCOUT_STATE_GEAROUT_WAITING_BUSY:
                               // Set next state
                               #statSyncOutState := #SYNCOUT_STATE_CHECK_ACTIVE;
                               #tempStateChangeActive := TRUE;

                             #SYNCOUT_STATE_GEAROUT_ACTIVE_BUSY:
                               #statSyncOutState := #SYNCOUT_STATE_DONE; // Set next state

                           END_CASE;
                           // Reset MC_Instruction
                           #instGearOut(Slave := #statAxis,
                                        Execute := FALSE);

                         ELSIF #instGearOut.CommandAborted THEN
                           #statSyncOutState := #SYNCOUT_STATE_ABORTED; // Set next state
                         END_IF;
                       END_REGION

                       // ===========================================================
                     #SYNCOUT_STATE_CAMOUT_WAITING_BUSY,
                     #SYNCOUT_STATE_CAMOUT_ACTIVE_BUSY:
                       REGION CAMOUT_BUSY
                         // Call MC_Instruction
                         #instCamOut(Slave := #statAxis,
                                     Execute := TRUE);

                         IF #instCamOut.Done THEN
                           CASE #statSyncOutState OF
                             #SYNCOUT_STATE_CAMOUT_WAITING_BUSY:
                               // Set next state
                               #statSyncOutState := #SYNCOUT_STATE_CHECK_ACTIVE;
                               #tempStateChangeActive := TRUE;

                             #SYNCOUT_STATE_CAMOUT_ACTIVE_BUSY:
                               #statSyncOutState := #SYNCOUT_STATE_DONE; // Set next state

                           END_CASE;
                           // Reset MC_Instruction
                           #instCamOut(Slave := #statAxis,
                                       Execute := FALSE);

                         ELSIF #instCamOut.CommandAborted THEN
                           #statSyncOutState := #SYNCOUT_STATE_ABORTED; // Set next state
                         END_IF;
                       END_REGION

                       // ===========================================================
                     #SYNCOUT_STATE_DONE,
                     #SYNCOUT_STATE_ABORTED,
                     #SYNCOUT_STATE_ERROR:
                       REGION FINISHED
                         IF NOT #statBasicCommand.%X11 THEN
                           // Return to NO_SELECTION if command finished
                           #statBasicMotionState := #NO_SELECTION;
                         END_IF;
                       END_REGION
                   END_CASE;

                   IF #instGearOut.Error THEN
                     // Errorhandling
                     #statStatus := #ERR_MC_GEAROUT;
                     #statStatusText := STRING#'ERR_MC_GEAROUT';
                     #statErrorAutoCleared := TRUE;
                     #statDiagnostics.subfunctionStatus := #statSubfunctionStatus := #instGearOut.ErrorID;
                     #statDiagnostics.basicMotionState := #statBasicMotionState;
                     #statFBState := #AXIS_STOP_ON_ERROR_SELECTION;
                     #statBasicMotionState := #NO_SELECTION;

                     #statSyncOutState := #SYNCOUT_STATE_ERROR; // Set next state

                   ELSIF #instCamOut.Error THEN
                     // Errorhandling
                     #statStatus := #ERR_MC_CAMOUT;
                     #statStatusText := STRING#'ERR_MC_CAMOUT';
                     #statErrorAutoCleared := TRUE;
                     #statDiagnostics.subfunctionStatus := #statSubfunctionStatus := #instCamOut.ErrorID;
                     #statDiagnostics.basicMotionState := #statBasicMotionState;
                     #statFBState := #AXIS_STOP_ON_ERROR_SELECTION;
                     #statBasicMotionState := #NO_SELECTION;

                     #statSyncOutState := #SYNCOUT_STATE_ERROR; // Set next state
                   END_IF;

                   // Write MC_Command outputs to internal variable
                   #statExeOfBasicMotion := 16#0;
                   #statExeOfBasicMotion.%X0 := #statSyncOutState < #SYNCOUT_STATE_DONE; // 7
                   #statExeOfBasicMotion.%X1 := #statSyncOutState = #SYNCOUT_STATE_DONE; // 7
                   #statExeOfBasicMotion.%X2 := #statSyncOutState = #SYNCOUT_STATE_ABORTED; // 8
                   #statExeOfBasicMotion.%X3 := #statSyncOutState = #SYNCOUT_STATE_ERROR; // 9
                   #statExeOfBasicMotion.%X6 := #instCamOut.StartSyncOut OR #instGearOut.StartSyncOut;
                 END_IF;
               END_REGION
             ELSE
               // Errorhandling
               #statStatus := #ERR_UNDEFINED_BASIC_MOTION_STATE;
               #statStatusText := STRING#'ERR_UNDEFINED_BASIC_MOTION_STATE';
               #statErrorUserCleared := TRUE;
               #statDiagnostics.subfunctionStatus := #statSubfunctionStatus := 0;
               // Set errorstate
               #statFBState := #FB_ERROR;
           END_CASE;
         #ABORT_WAITING_GEARINPOS_OR_CAMIN:
           // Abort waiting absolute gearing / camIn job if new basic motion job is selected (configuration.generalSettings.abortWaitingSyncCmd = TRUE)

           CASE #statWaitingFunctionStateAbortAutomatic OF
             #WFS_FS_GEARINPOS: // Waiting
               REGION GEARINPOS_WAITING
                 #instGearOut(Slave := #statAxis,
                              Execute := TRUE);

                 IF (#instGearOut.Done = TRUE) OR (#instGearOut.CommandAborted = TRUE)
                   //OR (LAxisCtrl_UnpubWaitingFunctionStateSyncAxis(#statAxis) = 0) // V1.1.0
                 THEN // Relative gearing command has aborted waiting absolute gearing job
                   #statMainSelectionState := #CALL_BASIC_MOTION; // Execute new basic motion command
                   #tempStateChangeActive := TRUE;
                   #statFirstCycleBasicMotion := TRUE;

                 ELSIF (#instGearOut.Error = TRUE)
                 THEN
                   #statStatus := #ERR_MC_GEAROUT;
                   #statStatusText := STRING#'ERR_MC_GEAROUT';
                   #statDiagnostics.subfunctionStatus := #statSubfunctionStatus := #instGearOut.ErrorID;
                   // Errorhandling
                   #statErrorAutoCleared := TRUE;
                   // Set next state
                   #statFBState := #AXIS_STOP_ON_ERROR_SELECTION;
                   #statMainSelectionState := #CALL_BASIC_MOTION;
                   #statBasicMotionState := #NO_SELECTION;
                 ELSE
                   ; // Command running
                 END_IF;

                 // Write MC_Command outputs to internal variable
                 #statExeOfBasicMotion := 16#0;
                 #statExeOfBasicMotion.%X0 := #instGearOut.Busy;
               END_REGION

             #WFS_FS_CAMIN: // Waiting
               REGION CAMIN_WAITING
                 #instCamOut(Slave := #statAxis,
                             Execute := TRUE);

                 IF (#instCamOut.Done = TRUE) OR (#instCamOut.CommandAborted = TRUE)
                   //OR (LAxisCtrl_UnpubWaitingFunctionStateSyncAxis(#statAxis) = 0) // V1.1.0
                 THEN
                   #statMainSelectionState := #CALL_BASIC_MOTION; // Execute new basic motion command
                   #tempStateChangeActive := TRUE;
                   #statFirstCycleBasicMotion := TRUE;

                 ELSIF (#instCamOut.Error = TRUE)
                 THEN
                   #statStatus := #ERR_MC_CAMOUT;
                   #statStatusText := STRING#'ERR_MC_CAMOUT';
                   #statDiagnostics.subfunctionStatus := #statSubfunctionStatus := #instCamOut.ErrorID;
                   // Errorhandling
                   #statErrorAutoCleared := TRUE;
                   // Set next state
                   #statFBState := #AXIS_STOP_ON_ERROR_SELECTION;
                   #statMainSelectionState := #CALL_BASIC_MOTION;
                   #statBasicMotionState := #NO_SELECTION;
                 ELSE
                   ; // Command running
                 END_IF;

                 // Write MC_Command outputs to internal variable
                 #statExeOfBasicMotion := 16#0;
                 #statExeOfBasicMotion.%X0 := #instCamOut.Busy;
               END_REGION

           END_CASE;
         ELSE
           // Errorhandling
           #statStatus := #ERR_UNDEFINED_MAIN_SELECTION_STATE;
           #statStatusText := STRING#'ERR_UNDEFINED_MAIN_SELECTION_STATE';
           #statErrorUserCleared := TRUE;
           #statDiagnostics.subfunctionStatus := #statSubfunctionStatus := 0;
           // Set errorstate
           #statFBState := #FB_ERROR;
       END_CASE;

     UNTIL (#tempStateChangeActive = FALSE)
     END_REPEAT;
   END_REGION

   //----------------------------------------------------------------------------------------------
   // Execution of homing functionality 
   //----------------------------------------------------------------------------------------------
   REGION EXECUTION_OF_PASSIVE_HOMING
     // Statemachine for homing functionality
     CASE #statPassiveHomingState OF
         // Selection of extended homing mode  
       #NO_HOMING_ACTIVE:
         ; // Do nothing

       #STANDARD_HOMING:
         // No additional features
         REGION STANDARD_HOMING
           // Firstcycle of command
           IF (#statFirstCycleHoming = TRUE) THEN
             // Reset MC_HOME command
             #instHome(Axis := #statAxis,
                       Execute := FALSE);
             IF (#statBasicMotionState = #ACTIVE_HOMING_SELECTED) THEN
               #statBasicMotionState := #NO_SELECTION;
             END_IF;
           END_IF;

           // Call MC_Command
           #instHome(Axis := #statAxis,
                     Execute := #statExtendedCommand.%X2, // Input: homing
                     Position := #configuration.homing.position,
                     Mode := #configuration.homing.mode);

           // Evaluate MC_Command
           IF (#instHome.Busy = FALSE) AND
             (#instHome.Done = FALSE) AND
             (#instHome.CommandAborted = FALSE) AND
             (#instHome.Error = FALSE)
           THEN
             // Return to NO_SELECTION if command finished
             #statPassiveHomingState := #NO_HOMING_ACTIVE;

           ELSIF (#instHome.Error = TRUE) THEN
             // Errorhandling
             #statStatus := #ERR_MC_HOME;
             #statStatusText := STRING#'ERR_MC_HOME';
             #statErrorAutoCleared := TRUE;
             #statDiagnostics.subfunctionStatus := #statSubfunctionStatus := #instHome.ErrorID;
             #statPassiveHomingState := #NO_HOMING_ACTIVE;
             // Set next state
             #statFBState := #AXIS_STOP_ON_ERROR_SELECTION;
           ELSE
             ; // Command selected
           END_IF;
           #statExeOfHoming := 16#0;
           #statExeOfHoming.%X0 := #instHome.Busy;
           #statExeOfHoming.%X1 := #instHome.Done;
           #statExeOfHoming.%X2 := #instHome.CommandAborted;
           #statExeOfHoming.%X3 := #instHome.Error;
         END_REGION
       ELSE
         // Errorhandling
         #statStatus := #ERR_INVALID_HOMING_EXTENDED_MODE;
         #statStatusText := STRING#'ERR_INVALID_HOMING_EXTENDED_MODE';
         #statErrorAutoCleared := TRUE;
         #statDiagnostics.subfunctionStatus := #statSubfunctionStatus := 0;
         #statDiagnostics.basicMotionState := #statBasicMotionState;
         #statDiagnostics.superimposedMotionState := #statSupImpMotionState;
         // Set next state
         #statFBState := #AXIS_STOP_ON_ERROR_SELECTION;
         #statBasicMotionState := #NO_SELECTION;
         #statPassiveHomingState := #NO_HOMING_ACTIVE;
     END_CASE;
   END_REGION

   //----------------------------------------------------------------------------------------------
   // Execution of functionalities of superimposed coordinate system
   //----------------------------------------------------------------------------------------------
   REGION EXECUTION_OF_SUPERIMPOSED_COMMANDS
     // Statemachine for superimposed motion commands
     // Write diagnostics
     #statDiagnostics.basicMotionState := #statBasicMotionState;
     #statDiagnostics.superimposedMotionState := #statSupImpMotionState;

     CASE #statSupImpMotionState OF
       #NO_SELECTION:
         ; // Do nothing

       #POS_SUPERIMPOSED_SELECTED:
         // Additional features (applicative) : Specified direction
         REGION POS_SUPERIMPOSED_SELECTED;
           // Firstcycle of command
           IF (#statFirstCycleSupImpMotion = TRUE) THEN
             // Configurate the direction of rotation
             IF ((#configuration.posSuperimposed.direction = 0) AND (#configuration.posSuperimposed.distance >= 0.0))  // Sign of distance is evaluated
               OR (#configuration.posSuperimposed.direction = #FORWARD_DIR)// Positive direction
             THEN
               #statSupImpMotionPosition := ABS(IN := #configuration.posSuperimposed.distance);
               // Reset MC_MOVESUPERIMPOSED command
               #instMoveSuperimposed(Axis := #statAxis,
                                     Execute := FALSE);
               #statApplicativeSupImpMotionError := FALSE;
             ELSIF ((#configuration.posSuperimposed.direction = 0) AND (#configuration.posSuperimposed.distance < 0.0)) // Sign of distance is evaluated
               OR (#configuration.posSuperimposed.direction = #BACKWARD_DIR)// Negative direction 
             THEN
               #statSupImpMotionPosition := - ABS(IN := #configuration.posSuperimposed.distance);
               // Reset MC_MOVESUPERIMPOSED command
               #instMoveSuperimposed(Axis := #statAxis,
                                     Execute := FALSE);
               #statApplicativeSupImpMotionError := FALSE;
             ELSE
               // Errorhandling - Invalid direction
               #statStatus := #ERR_INVALID_POS_SUPERIMPOSED_DIR;
               #statStatusText := STRING#'ERR_INVALID_POS_SUPERIMPOSED_DIR';
               #statErrorAutoCleared := TRUE;
               #statDiagnostics.subfunctionStatus := #statSubfunctionStatus := 0;
               #statApplicativeSupImpMotionError := TRUE;
               // Set next state
               #statFBState := #AXIS_STOP_ON_ERROR_SELECTION;
               #statSupImpMotionState := #NO_SELECTION;
             END_IF;
           END_IF;

           IF (#statApplicativeSupImpMotionError = FALSE) THEN
             // Call MC_Command
             #instMoveSuperimposed(Axis := #statAxis,
                                   Execute := #statSupImpCommand.%X0, // Input: posSuperimposed
                                   Distance := #statSupImpMotionPosition,
                                   VelocityDiff := #configuration.posSuperimposed.velocityDiff,
                                   Acceleration := #configuration.posSuperimposed.acceleration,
                                   Deceleration := #configuration.posSuperimposed.deceleration,
                                   Jerk := #configuration.posSuperimposed.jerk);

             // Evaluate MC_Command
             IF (#instMoveSuperimposed.Busy = FALSE) AND
               (#instMoveSuperimposed.Error = FALSE) AND
               (#instMoveSuperimposed.Done = FALSE) AND
               (#instMoveSuperimposed.CommandAborted = FALSE)
             THEN
               // Return to NO_SELECTION if command finished
               #statSupImpMotionState := #NO_SELECTION;

